FUNCTION_BLOCK DigitalOutput_HMI EXTENDS HmiFunction
VAR
	DigitalOutput : I_DigitalOutput;
	{ attribute 'TcHmiSymbol.AddSymbol' }
	{ attribute 'TcHmiSymbol.AddSymbol.UserGroups' := '__SystemAdministrators,Admin' }
	DigitalOutput_HMI : ST_DigitalOutput_HMI;
END_VAR

PROPERTY ControlObject : I_Base
SET
__QueryInterface(ControlObject,DigitalOutput);
END_SET
END_PROPERTY

METHOD CyclicLogic
IF DigitalOutput = 0 THEN
	RETURN;
END_IF

DigitalOutput_HMI.Name		 := DigitalOutput.Name;
DigitalOutput_HMI.On		 := DigitalOutput.On;
DigitalOutput_HMI.HmiEnabled := Enabled;
IF Enabled THEN
	DigitalOutput.Force := DigitalOutput_HMI.Force;
END_IF
END_METHOD

(*FB_Init is always available implicitly and it is used primarily for initialization.
The return value is not evaluated. For a specific influence, you can also declare the
methods explicitly and provide additional code there with the standard initialization
code. You can evaluate the return value.*)
METHOD FB_Init : BOOL
VAR_INPUT
	(* TRUE: the retain variables are initialized (reset warm / reset cold)*)
	bInitRetains : BOOL;

	(* TRUE: the instance will be copied to the copy code afterward (online change)   *)
	bInCopyCode	  : BOOL;
	Name		  : T_MaxString;
	DigitalOutput : I_DigitalOutput;
END_VAR
THIS^.DigitalOutput := DigitalOutput;
ControlType			:= 'DigitalOutput';
LinkObject			:= 'DigitalOutput_HMI';
END_METHOD

END_FUNCTION_BLOCK

(* stored: Version 1.1.0.1, ProductVersion 3.1.4026.18
   POU DigitalOutput_HMI: Id {f0113d82-f398-4272-9386-6b8d9f69409c}, SpecialFunc None
   Property ControlObject: Id {19cca1ad-4f51-4528-b3f2-3d0ff46c0e02}
   Set Set: Id {81ca5ed9-81a3-4253-813c-b7ed48c61998}
   Method CyclicLogic: Id {df85ed5d-381b-4deb-bcc1-ca5422013460}
   Method FB_Init: Id {9b4eb191-1358-471b-8dae-85cf149b3ce0} *)
